FUNCTION_BLOCK FB_Coordinador_SFC
VAR_IN_OUT
    UnidadesPendientes: UINT;
    UnidadesRealizadas: UINT;
END_VAR
VAR_INPUT
    // SFC-Flags
    SFCPause: BOOL;
    SFCReset: BOOL;
    
    // Indicadores de sincronizacion
    Ack: BOOL := TRUE;
    Execute: BOOL;
    
    // Parametros de sincronizacion
    PaleSituado: BOOL;
    BaseCargada: BOOL;
    RodamientoPrensado: BOOL;
    BaseDescargada: BOOL;
    PaleTransferido: BOOL;
    
    // Parametros
    CondicionInicial: BOOL;
    UnidadesSolicitadas: UINT;
END_VAR
VAR_OUTPUT
    // Indicadores de sincronizacion
    Done: BOOL;
    Ready: BOOL;

    // Parametros de sincronizacion
    SituaPale: BOOL;
    CargaBase: BOOL;
    PrensaRodamiento: BOOL;
    DescargaBase: BOOL;
    TransfierePale: BOOL;
    
    // Salidas
    LamparaAlarma: BOOL;
    LamparaMarcha: BOOL;
END_VAR
VAR
    // Bloques funcionales
    CLK: FB_Clock;
END_VAR

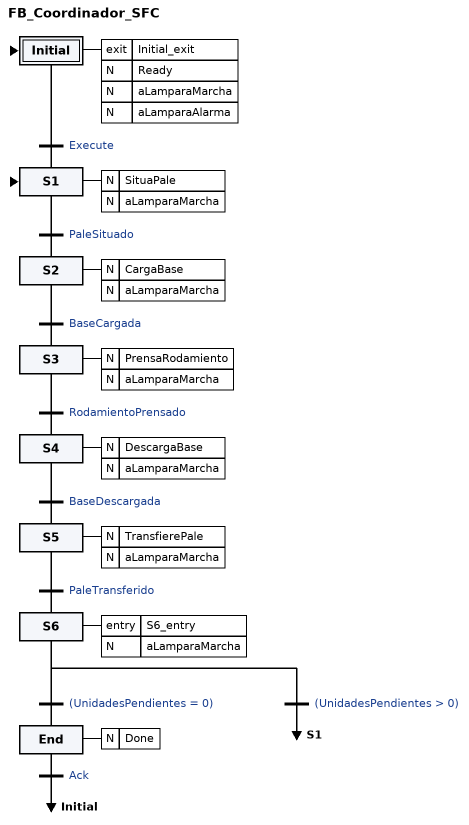
INITIAL_STEP Initial:
    Initial_exit(P0);  // exit action
    Ready(N);
    aLamparaMarcha(N);
    aLamparaAlarma(N);
END_STEP
TRANSITION FROM Initial TO S1
    := Execute;
END_TRANSITION
STEP S1:
    SituaPale(N);
    aLamparaMarcha(N);
END_STEP
TRANSITION FROM S1 TO S2
    := PaleSituado;
END_TRANSITION
STEP S2:
    CargaBase(N);
    aLamparaMarcha(N);
END_STEP
TRANSITION FROM S2 TO S3
    := BaseCargada;
END_TRANSITION
STEP S3:
    PrensaRodamiento(N);
    aLamparaMarcha(N);
END_STEP
TRANSITION FROM S3 TO S4
    := RodamientoPrensado;
END_TRANSITION
STEP S4:
    DescargaBase(N);
    aLamparaMarcha(N);
END_STEP
TRANSITION FROM S4 TO S5
    := BaseDescargada;
END_TRANSITION
STEP S5:
    TransfierePale(N);
    aLamparaMarcha(N);
END_STEP
TRANSITION FROM S5 TO S6
    := PaleTransferido;
END_TRANSITION
STEP S6:
    S6_entry(P1);  // entry action
    aLamparaMarcha(N);
END_STEP
TRANSITION FROM S6 TO End
    := (UnidadesPendientes = 0);
END_TRANSITION
TRANSITION FROM S6 TO S1
    := (UnidadesPendientes > 0);
END_TRANSITION
STEP End:
    Done(N);
END_STEP
TRANSITION FROM End TO Initial
    := Ack;
END_TRANSITION

ACTION aLamparaAlarma:
LamparaAlarma := (Initial.x AND NOT CondicionInicial AND CLK.Q);
END_ACTION

ACTION aLamparaMarcha:
LamparaMarcha := (Initial.x AND CondicionInicial AND CLK.Q) OR NOT Initial.x;

CLK();
END_ACTION

ACTION Initial_exit:
// Al iniciar una tarea se actualiza las unidades pendientes
IF (UnidadesPendientes = 0) THEN
    UnidadesPendientes := UnidadesSolicitadas;
END_IF
END_ACTION

ACTION S6_entry:
// Al completar la transferencia del pale
UnidadesRealizadas := UnidadesRealizadas + 1;

IF (UnidadesPendientes > 0) THEN
    UnidadesPendientes := UnidadesPendientes - 1;
END_IF
END_ACTION

END_FUNCTION_BLOCK

(* stored: Version 1.1.0.1, ProductVersion 3.1.4024.12
   POU FB_Coordinador_SFC: Id {91055dc8-8218-4ca0-bc1a-2b388a0f50ba}, SpecialFunc None
   Action aLamparaAlarma: Id {85868c8d-9492-454c-9a32-cd58bd12b035}
   Action aLamparaMarcha: Id {29376ebc-b13c-4e97-a81e-db432c3adea8}
   Action Initial_exit: Id {1d49c166-dc85-47eb-ba07-982d7526fd4f}
   Action S6_entry: Id {5da8d72d-fcf6-4f04-a27a-6abf8c70d5c7} *)
